Fanuc KAREL source: kd00060.KL

-- PROVISIONAL review KL for V940-1; original PC SHA256 e7bb84d0285a4593d4c405357208a87faf5503cf816459e3edf39b85defac1d0
-- Incomplete behavior may be omitted. Consult companion uncertainty JSON. Do not deploy.
PROGRAM KD00060
%NOLOCKGROUP
VAR
  I : INTEGER
  J : INTEGER
  B : BOOLEAN
  R : REAL
  S : STRING[80]
BEGIN
  -- V9_ZERO_TABLE_METADATA_HINT layout=0001; no indexed target words; source/name/runtime held
  -- UNRESOLVED_PC offsets 5-18; opcodes 9D,81,18,9D,1B,9D,12,9D,13,04
  -- UNRESOLVED_PC offsets 23-27; opcodes 7F
END KD00060
